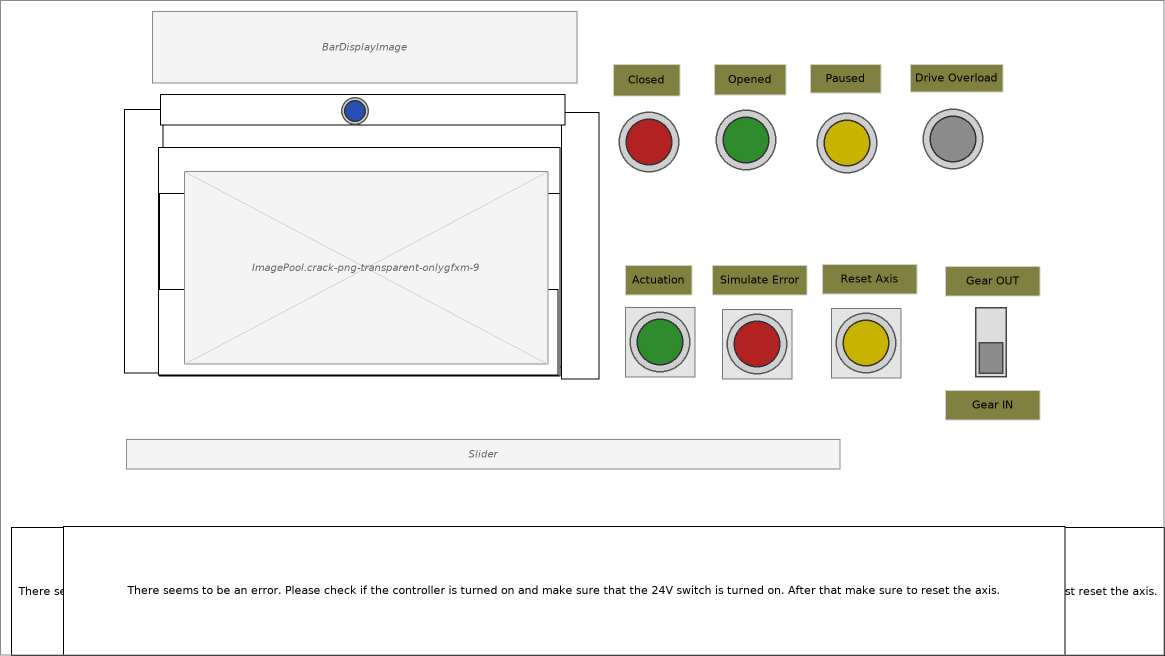
VISUALIZATION Visualization  // 1165x656
    Rectangle (161,123 402x244)
    Rectangle (124,109 39x264)
    Rectangle (561,112 38x267)
    Rectangle (160,94 405x31)
    Lamp1 (339,92 32x38), variable: GarageDoor.bMotionLight, style: Lamp-Lamp1-Blue
    Lamp1 (614,107 70x70), variable: GarageDoor.bDoorClosed, style: Lamp-Lamp1-Red
    Lamp1 (711,105 70x70), variable: GarageDoor.bDoorOpened, style: Lamp-Lamp1-Green
    Lamp1 (812,108 70x70), variable: GarageDoor.bDoorPaused, style: Lamp-Lamp1-Yellow
    Lamp1 (918,104 70x70), variable: GarageDoor.bDoorDriveOverload, style: Lamp-Lamp1-Gray
    PushSwitch (625,307 70x70), variable: GarageDoor.bActuationButton, behaviour: TAP, style: Switch-PushSwitch-Green
    PushSwitch (722,309 70x70), variable: GarageDoor.bErrorButton, behaviour: TAP, style: Switch-PushSwitch-Red
    Rectangle (161,274 399x96), invisible if: NOT GarageDoor.bTest1
    Rectangle (158,147 402x225), invisible if: NOT GarageDoor.bTest3
    Rectangle (160,205 399x166), invisible if: NOT GarageDoor.bTest2
    Rectangle (159,193 401x183), invisible if: NOT GarageDoor.bTest4
    Rectangle (158,289 400x86), invisible if: NOT GarageDoor.bTest5
    Image (184,171 364x193), invisible if: NOT GarageDoor.bErrorVis, image: ImagePool.crack-png-transparent-onlygfxm-9
    Textfield (613,64 67x32), "Closed", colour toggle: GarageDoor.bDoorClosed
    Textfield (714,64 72x31), "Opened", colour toggle: GarageDoor.bDoorOpened
    Textfield (810,64 71x29), "Paused", colour toggle: GarageDoor.bDoorPaused
    Textfield (910,64 93x28), "Drive Overload", colour toggle: GarageDoor.bDoorDriveOverload
    Textfield (625,265 67x30), "Actuation", colour toggle: GarageDoor.bActuationButton
    Textfield (712,265 95x30), "Simulate Error", colour toggle: GarageDoor.bErrorButton
    BarDisplayImage (152,11 425x72), value: GarageDoor.fPosition, style: BarDisplayImage-Gray, scale format: %.1f, scale 0..180
        p518627256: Axis Position
    PushSwitch (831,308 70x70), variable: GarageDoor.bResetButton, behaviour: TAP, style: Switch-PushSwitch-Yellow
    Textfield (822,264 95x30), "Reset Axis", colour toggle: GarageDoor.bErrorButton
    Rectangle (11,527 1154x129), "There seems to be an error. Please check if the resolver is connected properly and make sure that the power is turned on. After that make sure to reset the axis. If everything seems fine just reset the axis.", invisible if: NOT GarageDoor.bEncOrPwrErr
    Rectangle (63,526 1002x129), "There seems to be an error. Please check if the controller is turned on and make sure that the 24V switch is turned on. After that make sure to reset the axis.", invisible if: NOT GarageDoor.bCtrOr24VErr
    DipSwitch (956,307 70x70), variable: GarageDoor.bGearingButton, input disabled if: GarageDoor.bAxisMovement, behaviour: TOGGLE, style: Switch-DipSwitch-Gray
    Textfield (945,266 95x30), "Gear OUT", colour toggle: GarageDoor.bGearingButton
    Textfield (945,390 95x30), "Gear IN", colour toggle: NOT GarageDoor.bGearingButton
    Slider (126,439 714x30), variable: GarageDoor.rGearRatio, input disabled if: GarageDoor.bAxisMovement, scale 0..2
END_VISUALIZATION

(* stored: Version 1.1.0.1, ProductVersion 3.1.4024.12
   Visu Visualization: Id {76e93d4f-7cc7-4c37-872c-3d14c82ec7b2} *)
